PROGRAM RETURN_NG
VAR
	DELAY: TON;
END_VAR

IF NOT SORTER_VAR.I_NG_TRANSFER_AT_FRONT THEN
	SORTER_VAR.O_NG_DATA_OUTPUT1:=TRUE;
ELSE
	SORTER_VAR.O_NG_DATA_OUTPUT1:=FALSE;
END_IF

END_PROGRAM

(* stored: Version 1.1.0.1, ProductVersion 3.1.4020.12
   POU RETURN_NG: Id {328747e1-e495-488a-9c33-4bfcba7f10d1}, SpecialFunc None *)
